(* CODESYS project Manutec.project

Project tree, tasks and I/O mapping:
  Device : CODESYS SoftMotion Win V3, 3S - Smart Software Solutions GmbH, order no. 309021, version 3.5.9.20
    application Application
      libraries: VisuDialogs, * (System)
      task DefaultTask (cyclic, interval T#50ms, priority 16) calls Steuerung, Soll
      trace Sampling_Trace (task DefaultTask): Q1.ActPosition, Q1.ActVelocity, Steuerung.Rad1.MV
      global variables Globale_Variablen
      Visualization/
        visualisation FPL_Motor2
        visualisation FPL_PID
        visualisation Manutech
        visualisation FPL_SFC
      POUs/
        program Steuerung [FBD]
        function block TYP_Axis_MC [FBD]
        function block AddToAxesGroup [ST]
        function block DirectKin [ST]
        function block MoveDirectAbsolute [ST]
        function block ReverseKin [ST]
        function block SetKinTransform [FBD]
        program Ablauf [SFC]: Strecke2, Winkel3, Strecke3, Strecke4, Strecke1, Winkel4, Winkel1, Winkel2
        function block MoveLinearAbsolute [ST]
        program Soll [ST]
      data type AXES_GROUP_REF
      data type AXIS_REF
    SoftMotion General Axis Pool
      Drive1 : SM_Drive_Virtual, 3S - Smart Software Solutions GmbH, order no. 1805, version 4.0.0.0
          settings: fSWMaxVelocity = 1e3; fSWMaxAcceleration = 1e5; fSWMaxDeceleration = 1e5; fSWLimitNegative = -1000.0
      Drive2 : SM_Drive_Virtual, 3S - Smart Software Solutions GmbH, order no. 1805, version 4.0.0.0
          settings: fSWMaxVelocity = 1e3; fSWMaxAcceleration = 1e5; fSWMaxDeceleration = 1e5; fSWLimitNegative = -1000.0
      Drive3 : SM_Drive_Virtual, 3S - Smart Software Solutions GmbH, order no. 1805, version 4.0.0.0
          settings: wDriveID = 2; fSWMaxVelocity = 1e3; fSWMaxAcceleration = 1e5; fSWMaxDeceleration = 1e5; fSWLimitNegative = -1000.0
      Drive4 : SM_Drive_Virtual, 3S - Smart Software Solutions GmbH, order no. 1805, version 4.0.0.0
          settings: wDriveID = 3; fSWMaxVelocity = 1e3; fSWMaxAcceleration = 1e5; fSWMaxDeceleration = 1e5; fSWLimitNegative = -1000.0
      Drive5 : SM_Drive_Virtual, 3S - Smart Software Solutions GmbH, order no. 1805, version 4.0.0.0
          settings: wDriveID = 4; fSWMaxVelocity = 1e3; fSWMaxAcceleration = 1e5; fSWMaxDeceleration = 1e5; fSWLimitNegative = -1000.0
      Drive6 : SM_Drive_Virtual, 3S - Smart Software Solutions GmbH, order no. 1805, version 4.0.0.0
          settings: wDriveID = 5; fSWMaxVelocity = 1e3; fSWMaxAcceleration = 1e5; fSWMaxDeceleration = 1e5; fSWLimitNegative = -1000.0
  libraries: SysCallback23, 3.5.2.0 (System); Standard, 3.5.9.0 (System); VisuSymbols, 3.5.8.0 (System)
  text list GlobalTextList
*)

// Device/Application/AXES_GROUP_REF
TYPE AXES_GROUP_REF:
STRUCT
  Goal, pAbs:ARRAY[1..6] OF REAL;
  pRef, pAct:ARRAY[1..6] OF REAL;
  qRef, qAct:ARRAY[1..6] OF REAL;
  Go:BOOL;
  Done:BOOL;
  interpolating:BOOL;
END_STRUCT
END_TYPE

// Device/Application/AXIS_REF
TYPE AXIS_REF :
STRUCT
	qRef:REAL;
	vRef:REAL:=500;
	aRef:REAL:=300;
	SetPosition:REAL;
	SetVelocity:REAL;
	ActPosition:REAL;
	ActVelocity:REAL;
	Go, Stop, Reset, Error, Done:BOOL;
END_STRUCT
END_TYPE

// Device/Application/Globale_Variablen
VAR_GLOBAL CONSTANT
	PI: REAL := 3.141592654;
END_VAR
VAR_GLOBAL
	E0,E1 :DINT;
	A0 AT%QW0 :INT;
	A1 AT%QW1 :INT;
	A2 AT%QW2 :INT;
	A3 AT%QW3 :INT;
	Q1, Q2, Q3, Q4, Q5, Q6: AXIS_REF;
	Arm: AXES_GROUP_REF;
	Start, Stop, Reset, NotAus:BOOL;
	PtpMove: BOOL;
	LinMove: BOOL;
	Ziel: ARRAY [1..6] OF REAL;
	 l_0: REAL:=70.0;
     l_1: REAL:=70.0;
      l_2: REAL:=70.0;
	   
  l0: REAL:=0;									(* robot link lengths *)
  l1: REAL:=630;									
  l2: REAL:=350;								 
  l3: REAL:=350;									
  l5: REAL:=120; (*70;*)
  H:BOOL;
  
END_VAR

// Device/Application/POUs/Steuerung
PROGRAM Steuerung
VAR
	GroupAxis1,GroupAxis2,GroupAxis3,GroupAxis4,GroupAxis5,GroupAxis6:AddToAxesGroup;
	KinTransform: SetKinTransform;
	MoveDirect: MoveDirectAbsolute;
	MoveLinear: MoveLinearAbsolute;
	Achse1, Achse2, Achse3, Achse4, Achse5 ,Achse6: TYP_Axis_MC;
	
END_VAR

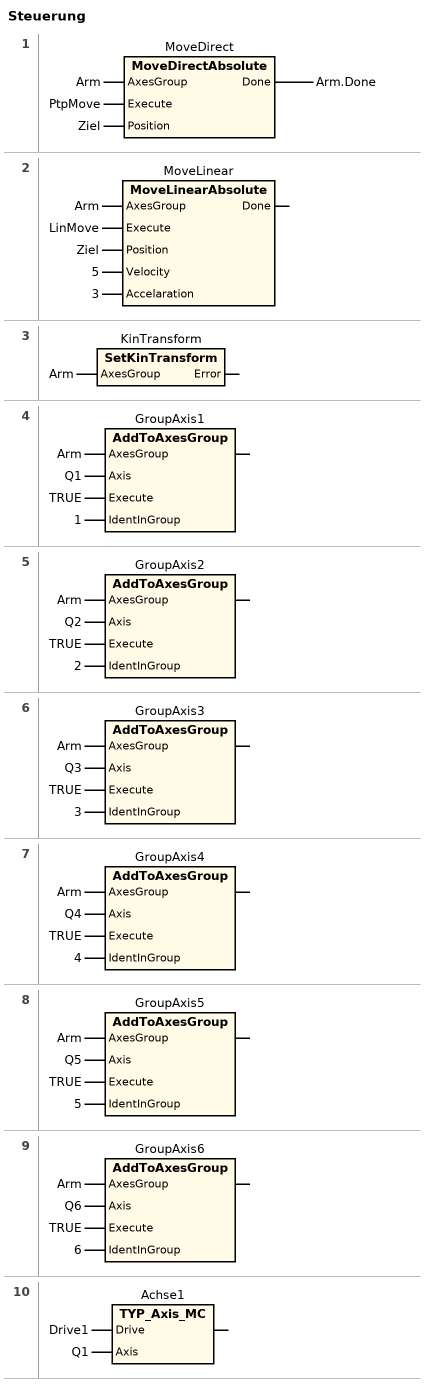
// NETWORK 1
MoveDirect(AxesGroup := Arm, Execute := PtpMove, Position := Ziel); // MoveDirectAbsolute
Arm.Done := MoveDirect.Done;

// NETWORK 2
MoveLinear(AxesGroup := Arm, Execute := LinMove, Position := Ziel, Velocity := 5, Accelaration := 3); // MoveLinearAbsolute

// NETWORK 3
KinTransform(AxesGroup := Arm); // SetKinTransform

// NETWORK 4
GroupAxis1(AxesGroup := Arm, Axis := Q1, Execute := TRUE, IdentInGroup := 1); // AddToAxesGroup

// NETWORK 5
GroupAxis2(AxesGroup := Arm, Axis := Q2, Execute := TRUE, IdentInGroup := 2); // AddToAxesGroup

// NETWORK 6
GroupAxis3(AxesGroup := Arm, Axis := Q3, Execute := TRUE, IdentInGroup := 3); // AddToAxesGroup

// NETWORK 7
GroupAxis4(AxesGroup := Arm, Axis := Q4, Execute := TRUE, IdentInGroup := 4); // AddToAxesGroup

// NETWORK 8
GroupAxis5(AxesGroup := Arm, Axis := Q5, Execute := TRUE, IdentInGroup := 5); // AddToAxesGroup

// NETWORK 9
GroupAxis6(AxesGroup := Arm, Axis := Q6, Execute := TRUE, IdentInGroup := 6); // AddToAxesGroup

// NETWORK 10
Achse1(Drive := Drive1, Axis := Q1); // TYP_Axis_MC

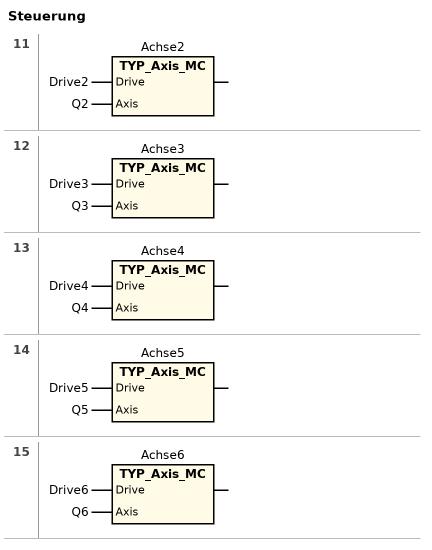
// NETWORK 11
Achse2(Drive := Drive2, Axis := Q2); // TYP_Axis_MC

// NETWORK 12
Achse3(Drive := Drive3, Axis := Q3); // TYP_Axis_MC

// NETWORK 13
Achse4(Drive := Drive4, Axis := Q4); // TYP_Axis_MC

// NETWORK 14
Achse5(Drive := Drive5, Axis := Q5); // TYP_Axis_MC

// NETWORK 15
Achse6(Drive := Drive6, Axis := Q6); // TYP_Axis_MC

END_PROGRAM

// Device/Application/POUs/MoveDirectAbsolute
FUNCTION_BLOCK MoveDirectAbsolute
VAR_IN_OUT 
  AxesGroup:AXES_GROUP_REF; (* Reference to a group of axes*) 
END_VAR
VAR_INPUT 
  Execute:  BOOL;  (*Start the motion at rising edge*) 
  Position:  ARRAY[1..6] OF REAL;
END_VAR
VAR_OUTPUT 
	Done: BOOL;
END_VAR
VAR
	eps:REAL:=0.1;
END_VAR

IF Execute THEN
	AxesGroup.Go:=1;
	AxesGroup.pRef[1]:=position[1];
	AxesGroup.pRef[2]:=position[2];
	AxesGroup.pRef[3]:=position[3];
	AxesGroup.pRef[4]:=position[4];
	AxesGroup.pRef[5]:=position[5];
	AxesGroup.pRef[6]:=position[6];
ELSE
	AxesGroup.Go:=0;
	Done:=0;
END_IF
IF 	ABS(AxesGroup.pAbs[1]-position[1])<eps AND
	ABS(AxesGroup.pAbs[2]-position[2])<eps AND
	ABS(AxesGroup.pAbs[3]-position[3])<eps AND
	ABS(AxesGroup.pAbs[4]-position[4])<eps AND
	ABS(AxesGroup.pAbs[5]-position[5])<eps AND
	ABS(AxesGroup.pAbs[6]-position[6])<eps THEN
  Done:=1;
END_IF

END_FUNCTION_BLOCK

// Device/Application/POUs/MoveLinearAbsolute
FUNCTION_BLOCK  MoveLinearAbsolute
VAR_IN_OUT 
  AxesGroup:AXES_GROUP_REF; (* Reference to a group of axes*) 
END_VAR
VAR_INPUT 
  Execute:  BOOL;  (*Start the motion at rising edge*) 
  Position:  ARRAY[1..6] OF REAL;
  Velocity:REAL;
  Accelaration:REAL;
END_VAR
VAR_OUTPUT 
  Done:  BOOL;  (* Commanded end positions reached FOR all axes*) 
END_VAR
VAR
    p_START:  ARRAY[1..6] OF LREAL;
	sp: LREAL;
	t, t1, t2, t3: LREAL;
	dist: LREAL;
	uhr: TP;
	EDGE: R_TRIG;
	Q: INT;
	ET: INT;
END_VAR

EDGE(CLK:=Execute);
 IF Edge.Q THEN
  p_Start[1]:=AxesGroup.pAct[1];
  p_Start[2]:=AxesGroup.pAct[2];
  p_Start[3]:=AxesGroup.pAct[3];
  AxesGroup.Done:=0;
 END_IF
 Dist:=SQRT(
			(Position[1]-p_Start[1])*(Position[1]-p_Start[1])+
			(Position[2]-p_Start[2])*(Position[2]-p_Start[2])+
            (Position[3]-p_Start[3])*(Position[3]-p_Start[3])
			);
 IF Dist>1 THEN
	Velocity:=LIMIT(0.001, Velocity, SQRT(Dist*Accelaration));		(* zeitoptimale Bahn *)
	t2:= Dist/Velocity;
	t1:= Velocity/Accelaration;
	t3:= t1+t2;
	uhr(IN:=Execute,pt:=LREAL_TO_TIME((t3+1)*1000));
	t:=TIME_TO_LREAL(uhr.ET)/1000;
	IF t < t1 THEN
		sp:= 0.5*Accelaration*t*t;
	ELSIF t >= t1 AND t<t2 THEN
		sp:= 0.5*Accelaration*t1*t1+ Velocity*(t-t1);
	ELSIF t >= t2 AND t<t3 THEN
		sp:= 0.5*Accelaration*t1*t1+ Velocity*(t2-t1)+ Velocity*(t-t2) - 0.5*Accelaration*(t-t2)*(t-t2);
	ELSIF t>=t3 THEN
		sp:= Dist;
		AxesGroup.Done:=1;
	END_IF
	IF execute THEN
		AxesGroup.pRef[1]:=p_START[1]+sp*(Position[1]-p_START[1])/Dist;
		AxesGroup.pRef[2]:=p_START[2]+sp*(Position[2]-p_START[2])/Dist;
		AxesGroup.pRef[3]:=p_START[3]+sp*(Position[3]-p_START[3])/Dist;
		AxesGroup.pRef[4]:= Position[4];
		AxesGroup.pRef[5]:= Position[5];
		AxesGroup.pRef[6]:= Position[6];
		
		
		
	END_IF	
	IF NOT Done THEN 
		AxesGroup.Go:=1;
	ELSE
		AxesGroup.Go:=0;
	END_IF
 END_IF

END_FUNCTION_BLOCK

// Device/Application/POUs/SetKinTransform
FUNCTION_BLOCK SetKinTransform
VAR_IN_OUT 
  AxesGroup:AXES_GROUP_REF; 
END_VAR
VAR_INPUT 
END_VAR
VAR_OUTPUT 
	Error:BOOL;
END_VAR
VAR
	IKT:ReverseKin;
	DKT:DirectKin;
	
END_VAR

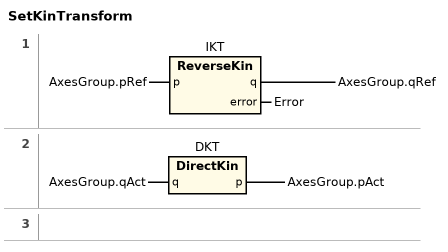
// NETWORK 1
IKT(p := AxesGroup.pRef, error => Error); // ReverseKin
AxesGroup.qRef := IKT.q;

// NETWORK 2
DKT(q := AxesGroup.qAct); // DirectKin
AxesGroup.pAct := DKT.p;

// NETWORK 3

END_FUNCTION_BLOCK

// Device/Application/POUs/ReverseKin
FUNCTION_BLOCK ReverseKin
VAR_INPUT
	p: ARRAY[1..6] OF REAL;
END_VAR
VAR_OUTPUT
	q: ARRAY[1..6] OF REAL;
	error: BOOL;
END_VAR
VAR
	rr: REAL;
	w:LREAL;
	alfa: REAL;
	beta: REAL;
	gamma: REAL;
	elbow_up:BOOL:=TRUE;
	X: REAL;
END_VAR

error:=FALSE;
IF ABS(p[1])<0.01 THEN p[1]:=0.01;
END_IF
q[1]:=ATAN(p[2]/p[1])*180/PI;

w:=SQRT(p[1]*p[1]+p[2]*p[2]);
IF ABS(w)<0.01 THEN w:=0.01;
END_IF
alfa:=ATAN((P[3]-l0-l1+l5)/w);

rr:= SQRT(w*w+(p[3]-l0-l1+l5)*(p[3]-l0-l1+l5));
IF ABS(rr)<0.01 THEN rr:=0.01;
END_IF
IF (l2+rr)<=l3 THEN beta:=PI;
  ELSIF ABS(l2-rr)>=l3 THEN beta:=0;
  ELSE beta:=ACOS((l2*l2+rr*rr-l3*l3)/(2*l2*rr));
END_IF
q[2]:=(alfa+beta)*180/PI;

IF (l2+l3)<=rr THEN gamma:=PI;
  ELSIF ABS(l2-l3)>=rr THEN gamma:=0;
  ELSE gamma:=ACOS((l2*l2-rr*rr+l3*l3)/(2*l2*l3));
END_IF
q[3]:=gamma*180/PI;
q[4]:=270-q[1]-q[2];
q[5]:=20;
q[6]:=30;


IF q[1]>80  OR q[1]<-80 OR q[2]>90  OR q[2]<0 OR q[3]>156  OR q[3]<65 OR q[4]>105  OR q[4]<20 OR  q[5]>20 OR q[5]<-20 OR q[6]>20  OR q[6]<-20  THEN error:=TRUE;
END_IF

END_FUNCTION_BLOCK

// Device/Application/POUs/DirectKin
FUNCTION_BLOCK DirectKin
VAR_INPUT
	q: ARRAY[1..6] OF REAL;         (*Axis angles*)
END_VAR
VAR_OUTPUT
	p: ARRAY[1..6] OF REAL;     (*Coordinates of the gripper*)
END_VAR
VAR
   oz,az,nz,nx,ny: REAL;
   
END_VAR

p[1]:= COS(q[1]*PI/180)*(l2*SIN(q[2]*PI/180)+ COS(q[2]*PI/180)*(SIN(q[3]*PI/180)*(l3+l5*COS(q[5]*PI/180))+l5*COS(q[3]*PI/180)*COS(q[4]*PI/180)*
	SIN(q[5]*PI/180))+ SIN(q[2]*PI/180)*( COS(q[3]*PI/180)*( l3+l5*COS(q[5]*PI/180))- l5*COS(q[4]*PI/180)*SIN(q[3]*PI/180)*SIN(q[5]*PI/180)))-
	l5*SIN(q[1]*PI/180)*SIN(q[4]*PI/180)*SIN(q[5]*PI/180);
	
p[2]:= -SIN(q[1]*PI/180)*(l2*SIN(q[2]*PI/180)+ COS(q[2]*PI/180)*(SIN(q[3]*PI/180)*(l3+l5*COS(q[5]*PI/180))+l5*COS(q[3]*PI/180)*COS(q[4]*PI/180)*
	SIN(q[5]*PI/180))+ SIN(q[2]*PI/180)*( COS(q[3]*PI/180)*( l3+l5*COS(q[5]*PI/180))- l5*COS(q[4]*PI/180)*SIN(q[3]*PI/180)*SIN(q[5]*PI/180)))-
	l5*COS(q[1]*PI/180)*SIN(q[4]*PI/180)*SIN(q[5]*PI/180);
	
p[3]:= l1+l2*COS(q[2]*PI/180)+ COS(q[2]*PI/180)*(COS(q[3]*PI/180)*(l3+l5*COS(q[5]*PI/180))-l5*COS(q[4]*PI/180)*SIN(q[3]*PI/180)*
	SIN(q[5]*PI/180))- SIN(q[2]*PI/180)*(SIN(q[3]*PI/180)*(l3+l5*COS(q[5]*PI/180))+l5*COS(q[3]*PI/180)*COS(q[4]*PI/180)*
	SIN(q[5]*PI/180));

oz:= -COS(q[2]*PI/180)*(SIN(q[3]*PI/180)*(COS(q[6]*PI/180)*SIN(q[4]*PI/180)+ COS(q[4]*PI/180)*COS(q[5]*PI/180)*SIN(q[6]*PI/180))+ 
    COS(q[3]*PI/180)*SIN(q[5]*PI/180)*SIN(q[6]*PI/180))- SIN(q[2]*PI/180)*(COS(q[3]*PI/180)*(COS(q[6]*PI/180)*SIN(q[4]*PI/180)+
    COS(q[4]*PI/180)*COS(q[5]*PI/180)*SIN(q[6]*PI/180))- SIN(q[3]*PI/180)*SIN(q[5]*PI/180)*SIN(q[6]*PI/180));
az:= COS(q[2]*PI/180)*(COS(q[3]*PI/180)*COS(q[5]*PI/180)- COS(q[4]*PI/180)*SIN(q[3]*PI/180)*SIN(q[5]*PI/180))- SIN(q[2]*PI/180)*(
    COS(q[5]*PI/180)*SIN(q[3]*PI/180)+COS(q[3]*PI/180)*COS(q[4]*PI/180)*SIN(q[5]*PI/180));

IF az>0 THEN p[4]:= ATAN(oz/az);
ELSIF az<0 THEN p[4]:=ATAN(oz/az)+PI;
	ELSIF az=0 AND oz>0 THEN p[4]:=1;
		ELSIF az=0 AND oz<0 THEN p[4]:=-1;
			ELSE P[4]:=0;
END_IF
 

nz:= COS(q[2]*PI/180)*(SIN(q[3]*PI/180)*( SIN(q[4]*PI/180)*SIN(q[6]*PI/180)-COS(q[4]*PI/180)*COS(q[5]*PI/180)*COS(q[6]*PI/180))-
    COS(q[3]*PI/180)*COS(q[5]*PI/180)*SIN(q[5]*PI/180))+ SIN(q[2]*PI/180)*(COS(q[3]*PI/180)*(SIN(q[4]*PI/180)*SIN(q[6]*PI/180)-
    COS(q[4]*PI/180)*COS(q[5]*PI/180)*COS(q[6]*PI/180))+ COS(q[6]*PI/180)*SIN(q[3]*PI/180)*SIN(q[5]*PI/180));
nx:=-COS(q[4]*PI/180)*(COS(q[2]*PI/180)*(COS(q[3]*PI/180)*(SIN(q[4]*PI/180)*SIN(q[6]*PI/180)-COS(q[4]*PI/180)*COS(q[5]*PI/180)*
    COS(q[6]*PI/180))- COS(q[6]*PI/180)*SIN(q[3]*PI/180)*SIN(q[5]*PI/180))-SIN(q[2]*PI/180)*(SIN(q[3]*PI/180)*(SIN(q[4]*PI/180)*SIN(q[6]*PI/180)-COS(q[4]*PI/180)*COS(q[5]*PI/180)*
    COS(q[6]*PI/180))- COS(q[3]*PI/180)*COS(q[6]*PI/180)*SIN(q[5]*PI/180)))-SIN(q[1]*PI/180)*(COS(q[4]*PI/180)*SIN(q[6]*PI/180)+
	COS(q[5]*PI/180)*COS(q[6]*PI/180)*SIN(q[4]*PI/180));
ny:= SIN(q[1]*PI/180)*(COS(q[2]*PI/180)*(COS(q[3]*PI/180)*(SIN(q[4]*PI/180)*SIN(q[6]*PI/180)-COS(q[4]*PI/180)*COS(q[5]*PI/180)*
    COS(q[6]*PI/180))- COS(q[6]*PI/180)*SIN(q[3]*PI/180)*SIN(q[5]*PI/180))-SIN(q[2]*PI/180)*(SIN(q[3]*PI/180)*(SIN(q[4]*PI/180)*SIN(q[6]*PI/180)-COS(q[4]*PI/180)*COS(q[5]*PI/180)*
    COS(q[6]*PI/180))- COS(q[3]*PI/180)*COS(q[6]*PI/180)*SIN(q[5]*PI/180)))-COS(q[1]*PI/180)*(COS(q[4]*PI/180)*SIN(q[6]*PI/180)+
	COS(q[5]*PI/180)*COS(q[6]*PI/180)*SIN(q[4]*PI/180));

P[5]:= ATAN(nz/SQRT((nx*nx)*(ny*ny)));

IF nx>0 THEN p[6]:= ATAN(ny/nx);
ELSIF nx<0 THEN p[6]:=ATAN(ny/nx)+PI;
	ELSIF nx=0 AND ny>0 THEN p[6]:=1;
		ELSIF nx=0 AND ny<0 THEN p[6]:=-1;
			ELSE P[6]:=0;
END_IF

END_FUNCTION_BLOCK

// Device/Application/POUs/AddToAxesGroup
FUNCTION_BLOCK AddToAxesGroup
VAR_IN_OUT 
  AxesGroup:AXES_GROUP_REF; (* Reference to a group of axes*) 
  Axis:AXIS_REF;
END_VAR
VAR_INPUT 
  Execute:  BOOL;  (*Start the motion at rising edge*) 
  IdentInGroup:  INT;
END_VAR
VAR_OUTPUT 
END_VAR
VAR
END_VAR

IF Execute THEN
   Axis.qRef:=AxesGroup.qRef[IdentInGroup];
   AxesGroup.qAct[IdentInGroup]:=Axis.ActPosition;
   Axis.Go:=AxesGroup.Go;
END_IF

END_FUNCTION_BLOCK

// Device/Application/POUs/TYP_Axis_MC
FUNCTION_BLOCK TYP_Axis_MC
VAR_IN_OUT
	Drive: AXIS_REF_SM3;
	Axis: AXIS_REF;
END_VAR
VAR_INPUT
END_VAR
VAR_OUTPUT
END_VAR
VAR
	MoveAbsolute: MC_MoveAbsolute;
	Power: MC_Power;
	ResetAxis:MC_SetPosition;
	MC_GroupHalt_0: MC_GroupHalt;
	D:AXIS_Group_REF_SM3;
END_VAR

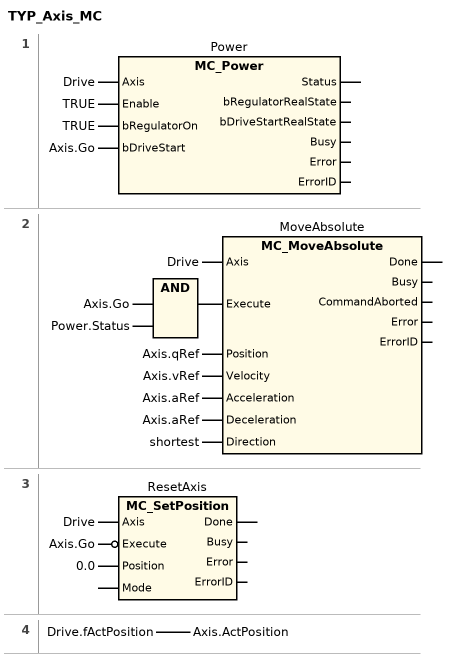
// NETWORK 1
Power(Axis := Drive, Enable := TRUE, bRegulatorOn := TRUE, bDriveStart := Axis.Go); // MC_Power

// NETWORK 2
MoveAbsolute(
    Axis := Drive,
    Execute := Axis.Go AND Power.Status,
    Position := Axis.qRef,
    Velocity := Axis.vRef,
    Acceleration := Axis.aRef,
    Deceleration := Axis.aRef,
    Direction := shortest); // MC_MoveAbsolute

// NETWORK 3
ResetAxis(Axis := Drive, Execute := NOT Axis.Go, Position := 0.0); // MC_SetPosition

// NETWORK 4
Axis.ActPosition := Drive.fActPosition;

END_FUNCTION_BLOCK

// Device/Application/POUs/Soll
PROGRAM Soll
VAR
	
END_VAR

Ziel[1]:= 50;
Ziel[2]:= 40;
Ziel[3]:= 60;
Ziel[4]:= 180;
Ziel[5]:= 0;
Ziel[6]:= 180;

END_PROGRAM

// Device/Application/POUs/Ablauf
PROGRAM Ablauf
VAR
	Path: ARRAY[1..4,1..2] OF REAL :=[ 	100,0,100,50,0,50, 0,0];
	SFCCurrentStep:STRING; (*Name des aktuellen Schritts*)
	TIPP:BOOL;
END_VAR

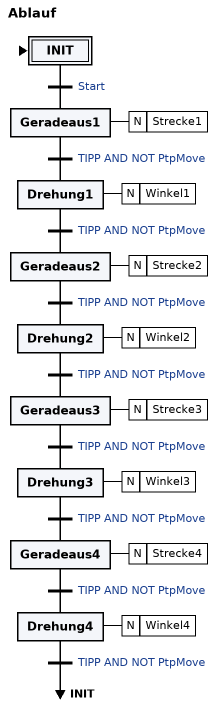
INITIAL_STEP INIT:
END_STEP
TRANSITION FROM INIT TO Geradeaus1
    := Start;
END_TRANSITION
STEP Geradeaus1:  // min time t#1s
    Strecke1(N);
END_STEP
TRANSITION FROM Geradeaus1 TO Drehung1
    := TIPP AND NOT PtpMove;
END_TRANSITION
STEP Drehung1:  // min time t#1s
    Winkel1(N);
END_STEP
TRANSITION FROM Drehung1 TO Geradeaus2
    := TIPP AND NOT PtpMove;
END_TRANSITION
STEP Geradeaus2:  // min time t#1s
    Strecke2(N);
END_STEP
TRANSITION FROM Geradeaus2 TO Drehung2
    := TIPP AND NOT PtpMove;
END_TRANSITION
STEP Drehung2:  // min time t#1s
    Winkel2(N);
END_STEP
TRANSITION FROM Drehung2 TO Geradeaus3
    := TIPP AND NOT PtpMove;
END_TRANSITION
STEP Geradeaus3:  // min time t#1s
    Strecke3(N);
END_STEP
TRANSITION FROM Geradeaus3 TO Drehung3
    := TIPP AND NOT PtpMove;
END_TRANSITION
STEP Drehung3:  // min time t#1s
    Winkel3(N);
END_STEP
TRANSITION FROM Drehung3 TO Geradeaus4
    := TIPP AND NOT PtpMove;
END_TRANSITION
STEP Geradeaus4:  // min time t#1s
    Strecke4(N);
END_STEP
TRANSITION FROM Geradeaus4 TO Drehung4
    := TIPP AND NOT PtpMove;
END_TRANSITION
STEP Drehung4:  // min time t#1s
    Winkel4(N);
END_STEP
TRANSITION FROM Drehung4 TO INIT
    := TIPP AND NOT PtpMove;
END_TRANSITION

ACTION Strecke2:
Ziel[1]:=Path[2,1];
Ziel[2]:=Path[2,2];
END_ACTION

ACTION Winkel3:
Ziel[6]:=270;
END_ACTION

ACTION Strecke3:
Ziel[1]:=Path[3,1];
Ziel[2]:=Path[3,2];
END_ACTION

ACTION Strecke4:
Ziel[1]:=Path[4,1];
Ziel[2]:=Path[4,2];
END_ACTION

ACTION Strecke1:
Ziel[1]:=Path[1,1];
Ziel[2]:=Path[1,2];
END_ACTION

ACTION Winkel4:
Ziel[6]:=360;
END_ACTION

ACTION Winkel1:
Ziel[6]:=90;
END_ACTION

ACTION Winkel2:
Ziel[6]:=180;
END_ACTION

END_PROGRAM

// Device/Application/Visualization/FPL_Motor2
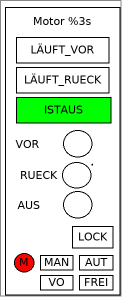
VISUALIZATION FPL_Motor2  // 122x297
VAR_INPUT
	Name: STRING;
END_VAR
VAR_IN_OUT
	IDF:TYP_IDF2;
END_VAR
    RoundedRectangle (92,133 0x0)
    Rectangle (5,7 115x288)
    Ellipse (15,133 27x23), "VOR"
    Rectangle (16,37 93x26), "LÄUFT_VOR", colour toggle: IDF.OUT1
    Rectangle (15,194 28x23), "AUS"
    Rectangle (16,97 95x26), "ISTAUS", colour toggle: IDF.OUT1 OR IDF.OUT2
    Ellipse (63,130 29x27), colour toggle: IDF.MAN_ON1
        tap IDF.MAN_ON1
    Ellipse (63,191 29x27), colour toggle: IDF.MAN_OFF
        tap IDF.MAN_OFF
    Ellipse (13,10 98x23), "Motor %3s", text variable: Name
    Rectangle (16,67 93x26), "LÄUFT_RUECK", colour toggle: IDF.OUT2
    RoundedRectangle (92,164 0x0)
    Ellipse (14,164 46x23), "RUECK"
    Ellipse (62,162 29x26), colour toggle: IDF.MAN_ON2
        tap IDF.MAN_ON2
    RoundedRectangle (72,226 41x22), "LOCK", colour toggle: IDF.LOCK1 oR IDF.LOCK2
    Rectangle (79,255 34x15), "AUT", colour toggle: IDF.AUT
    Rectangle (40,255 33x15), "MAN", colour toggle: IDF.MAN
    Ellipse (14,253 20x19), "M", colour toggle: IDF.SEL_MAN
        toggle IDF.SEL_MAN
    Rectangle (40,275 33x15), "VO", colour toggle: IDF.sel_MODE.LOCAL
    Rectangle (79,275 34x15), "FREI", colour toggle: IDF.SEL_MODE.FREE
END_VISUALIZATION

// Device/Application/Visualization/FPL_PID
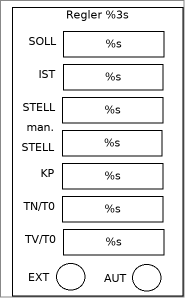
VISUALIZATION FPL_PID  // 185x298
VAR_INPUT
	Name: STRING;
END_VAR
VAR_IN_OUT
	Contr:TYP_PID;
END_VAR
    Rectangle (12,7 171x289), "Regler %3s", text variable: Name
    Rectangle (25,266 27x23), "EXT"
    Ellipse (56,263 29x27), colour toggle: Contr.ext
        toggle Contr.EXT
    Rectangle (63,31 101x26), "%s", text variable: Contr.w
        OnMouseDown: write Contr.Ref via Edit
    Rectangle (63,64 100x26), "%s", text variable: Contr.PV
    Ellipse (25,30 34x23), "SOLL"
    Ellipse (24,63 34x23), "IST"
    Ellipse (102,267 27x23), "AUT"
    Ellipse (132,264 29x27), colour toggle: Contr.AUT
        toggle Contr.AUT
    Rectangle (62,97 101x26), "%s", text variable: Contr.MV
    Rectangle (62,130 100x26), "%s", text variable: Contr.MV_MAN
        OnMouseDown: write Contr.MV_MAN via Default
    Ellipse (17,96 41x23), "STELL"
    Ellipse (18,136 39x23), "STELL"
    Ellipse (16,116 41x23), "man."
    Ellipse (23,162 34x23), "KP"
    Ellipse (24,195 34x23), "TN/T0"
    Ellipse (25,228 34x23), "TV/T0"
    Rectangle (62,163 101x26), "%s", text variable: Contr.KP
        OnMouseDown: write Contr.KP via Edit
    Rectangle (62,196 101x26), "%s", text variable: Contr.TN_T0
        OnMouseDown: write Contr.TN_T0 via Edit
    Rectangle (63,229 101x26), "%s", text variable: Contr.TV_T0
        OnMouseDown: write Contr.TV_T0 via Edit
END_VISUALIZATION

// Device/Application/Visualization/Manutech
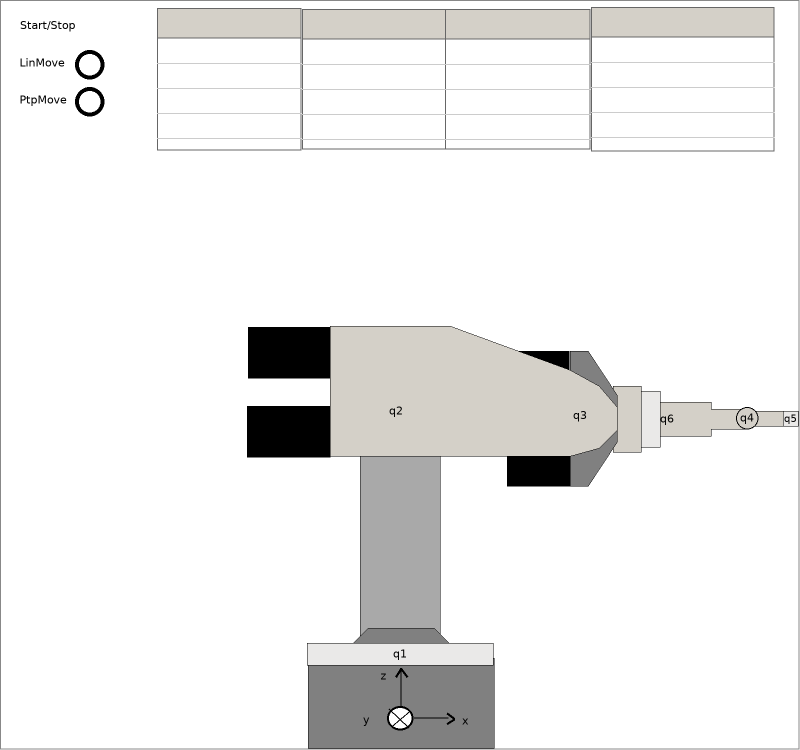
VISUALIZATION Manutech  // 800x750
    Rectangle (127,5 20x20)
    RoundedRectangle (17,14 72x23), "Start/Stop"
    Ellipse (75,50 29x29), colour toggle: LinMove
        toggle LinMove
    RoundedRectangle (13,40 55x46), "LinMove"
    Ellipse (75,87 29x29), colour toggle: PtpMove
        toggle PtpMove
    RoundedRectangle (15,77 55x46), "PtpMove"
    Polygon (360,419) (360,644) (440,644) (440,419)
    Polygon (308,748) (308,658) (338,658) (368,628) (434,628) (464,658) (494,658) (494,748)
    Polygon (307,643) (307,665) (493,665) (493,643), "q1"
    Polygon (505,351) (505,382) (569,382) (569,351)
        p2858320360: Arm.pRef[2]
        p3560616238: -175*(1-cos((Arm.pRef[1])*(3.14/180)))
        p2738717112: -175*(sin((180+Arm.pRef[1])*(3.14/180)))
    Polygon (507,455) (507,486) (571,486) (571,455)
        p2858320360: Arm.pRef[2]
        p3560616238: -175*(1-cos((Arm.pRef[1])*(3.14/180)))
        p2738717112: -175*(sin((180+Arm.pRef[1])*(3.14/180)))
    Polygon (489,403) (489,434) (553,434) (553,403)
        p2858320360: Arm.pRef[2]
        p3560616238: -175*(1-cos((Arm.pRef[1])*(3.14/180)))
        p2738717112: -175*(sin((180+Arm.pRef[1])*(3.14/180)))
    Polygon (247,406) (247,457) (330,457) (330,406)
        p2858320360: Arm.pRef[1]
    Polygon (248,327) (248,378) (331,378) (331,327)
        p2858320360: Arm.pRef[1]
    Ellipse (387,706 26x24)
    Line (401,707) (401,670)
    Polyline (396,677) (401,669) (407,677)
    Line (448,718) (414,718)
    Polyline (447,713) (455,719) (447,724)
    Rectangle (455,711 21x20), "x"
    Rectangle (353,710 27x20), "y"
    Rectangle (373,666 21x20), "z"
    Polygon (748,411) (750,426) (783,426) (783,411)
        p3560616238: (-175*(1-cos((Arm.pRef[1])*(3.14/180)))-173*(1-cos(((Arm.pRef[1])+Arm.pRef[2])*(3.14/180))))
        p2738717112: (173*sin((Arm.pRef[1]+Arm.pRef[2])*(3.14/180))+175*sin((Arm.pRef[1])*(3.14/180)))
        p2858320360: Arm.pRef[1] + Arm.pRef[2]+ 40
    Polygon (589,419) (613,400) (613,386) (641,386) (641,391) (660,391) (660,402) (711,402) (711,409) (745,409) (745,429) (711,429) (711,436) (660,436) (660,447) (641,447) (641,452) (613,452) (613,438), "q6"
        p3560616238: -175*(1-cos((Arm.pRef[1])*(3.14/180)))
        p2738717112: -175*sin((180+Arm.pRef[1])*(3.14/180))
        p2858320360: (Arm.pRef[1]+Arm.pRef[2])
    Ellipse (736,407 22x22), "q4"
        p3560616238: -175*(1-cos((Arm.pRef[1])*(3.14/180)))
        p2738717112: -175*sin((180+Arm.pRef[1])*(3.14/180))
        p2277200375: (Arm.pRef[1]+Arm.pRef[2])
    Polygon (783,411) (783,426) (798,426) (798,411), "q5"
        p3560616238: (-175*(1-cos((Arm.pRef[1])*(3.14/180)))-173*(1-cos(((Arm.pRef[1])+Arm.pRef[2])*(3.14/180))))
        p2738717112: (173*sin((Arm.pRef[1]+Arm.pRef[2])*(3.14/180))+175*sin((Arm.pRef[1])*(3.14/180)))
        p2858320360: Arm.pRef[1]+Arm.pRef[2]+40
    Table (157,8 144x142), data array: Arm.pRef
        p3854506369: Arm.pRef[INDEX]
    Table (302,9 144x140), data array: Arm.pAct
        p3854506369: Arm.pAct[INDEX]
    Table (445,9 145x140), data array: Arm.qAct
        p3854506369: Arm.qAct[INDEX]
    Table (591,7 183x144), data array: Arm.qRef
        p3854506369: Arm.qRef[INDEX]
    Polygon (641,391) (641,447) (660,447) (660,391)
        p3560616238: -175*(1-cos((Arm.pRef[1])*(3.14/180)))
        p2738717112: -175*sin((180+Arm.pRef[1])*(3.14/180))
        p2858320360: ( Arm.pRef[1]+ Arm.pRef[2] )
    Polygon (617,395) (617,442) (588,486) (570,486) (570,351) (588,351)
        p2858320360: Arm.pRef[2]
        p3560616238: -175*(1-cos((Arm.pRef[1])*(3.14/180)))
        p2738717112: -175*(sin((180+Arm.pRef[1])*(3.14/180)))
    Polygon (330,326) (330,456) (570,456) (599,448) (617,430) (617,407) (599,386) (570,370) (450,326)
        p2858320360: Arm.pRef[1]
    Label (349,395 94x32), "q2"
    Polygon (569,404) (569,427) (591,427) (591,404) (591,404), "q3"
        p2858320360: Arm.pRef[1]
    Line (410,711) (391,727)
    Line (409,728) (389,709)
END_VISUALIZATION

// Device/Application/Visualization/FPL_SFC
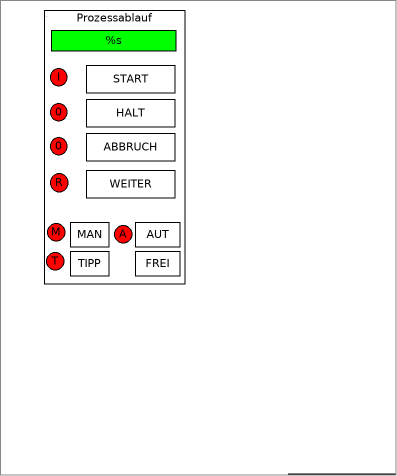
VISUALIZATION FPL_SFC  // 397x476
    Rectangle (288,474 107x0)
    Rectangle (44,10 141x274), "Prozessablauf", colour toggle: Ablauf .STOP
    Ellipse (46,16 0x0)
    Ellipse (50,173 18x19), "R", colour toggle: Ablauf.WEITER
        tap Ablauf.WEITER
    Rectangle (51,30 125x21), "%s", text variable: Ablauf.SFCCurrentStep
    Rectangle (86,99 89x28), "HALT", colour toggle: Ablauf.HALT
    Ellipse (46,252 18x18), "T", colour toggle: Ablauf.SEL_TIPP
        toggle Ablauf.SEL_TIPP
    Rectangle (70,222 39x25), "MAN", colour toggle: Ablauf .MAN
    Rectangle (70,251 39x25), "TIPP", colour toggle: Ablauf.TIPP
    Rectangle (135,222 45x25), "AUT", colour toggle: Ablauf.AUT
    Rectangle (135,251 45x25), "FREI", colour toggle: Ablauf.Frei
    Ellipse (50,68 17x18), "I", colour toggle: Ablauf.START
        tap Ablauf.START
    Rectangle (86,65 89x28), "START", colour toggle: Ablauf.START
    Rectangle (86,170 89x28), "WEITER", colour toggle: Ablauf.WEITER
    Ellipse (50,103 17x18), "0", colour toggle: Ablauf.HALT
        tap Ablauf.HALT
    Rectangle (86,133 89x28), "ABBRUCH", colour toggle: Ablauf.ABBRUCH
    Ellipse (50,137 17x18), "0", colour toggle: Ablauf.ABBRUCH
        tap Ablauf.ABBRUCH
    Ellipse (47,223 18x18), "M", colour toggle: Ablauf.SEL_MAN
        toggle Ablauf.SEL_MAN
    Ellipse (114,225 18x18), "A", colour toggle: Ablauf.SEL_AUT
        toggle Ablauf.SEL_AUT
END_VISUALIZATION
